FUNCTION_BLOCK Gripper
VAR
	Close	: BOOL;
	Closed	: BOOL;
	Opened 	: BOOL;
END_VAR

METHOD mClose : BOOL
VAR_INPUT
END_VAR
//IF ActInputs.Opened AND Flags.PartReady THEN (Faulty)
//	Close := ActOutputs.Close := TRUE;
//END_IF

Close := TRUE;
END_METHOD

METHOD mClosed : BOOL
VAR_INPUT
END_VAR
END_METHOD

METHOD mOpened : BOOL
VAR_INPUT
END_VAR
END_METHOD

PROPERTY pClose : BOOL
GET
pClose := Close;
END_GET
SET
Close := pClose;
END_SET
END_PROPERTY

PROPERTY pClosed : BOOL
GET
pClosed := Closed;
END_GET
SET
Closed := pClosed;
END_SET
END_PROPERTY

PROPERTY pOpened : BOOL
GET
END_GET
SET
END_SET
END_PROPERTY

END_FUNCTION_BLOCK

(* stored: Version 1.1.0.1, ProductVersion 3.1.4024.9
   POU Gripper: Id {e2e07011-251c-448f-bd09-229b297fbd8e}, SpecialFunc None
   Method mClose: Id {17dccae4-20dd-4877-98db-cf4ed4a6c5e2}
   Method mClosed: Id {11b78d51-ee76-4a45-b2f1-5569cce0e23b}
   Method mOpened: Id {de9fb022-6787-414b-ad8e-01d419699a7b}
   Property pClose: Id {812aa284-5443-43fb-bb05-4314027d3207}
   Get Get: Id {cd4d5a53-ba36-43a2-9efe-e7b681f38d55}
   Set Set: Id {7e809eb5-b39b-4d9b-a1f8-54a4ced74be3}
   Property pClosed: Id {87702b9a-bcde-4702-9221-05b3ca2875e2}
   Get Get: Id {0c581010-4917-41b2-b3d8-7a46fa1a1336}
   Set Set: Id {d7dfec96-1d27-4aee-940f-c68e7c0bdc53}
   Property pOpened: Id {fb91f2b5-5c93-409c-b5d0-217de858f212}
   Get Get: Id {4d5d8842-7b40-4832-84e8-ba9231c21e5f}
   Set Set: Id {0ecad2ea-6889-4db8-8f2f-0416b723b4b7} *)
